// TIA Portal V19 export
DATA_BLOCK "FILL DB"   // DB999
{ S7_Optimized_Access := 'TRUE' }
// stored: AutoNumber false, MemoryReserve 0
   VAR RETAIN
      FILL : Array[0..31] of Int;
   END_VAR
BEGIN
   FILL[0..31] := 9999;
END_DATA_BLOCK
